TYPE E_RolloMode : (
	eRollo_Stop,
	eRollo_Manuell,
	eRollo_Auto,
	eRollo_Schatten);
END_TYPE

(* stored: Version 1.1.0.1, ProductVersion 3.1.4018.5
   DUT E_RolloMode: Id {d807219a-a737-4ff7-bb9e-10e735a825b7} *)
